INTERFACE I_NodeExecuteBeginEvent EXTENDS I_Event

PROPERTY PUBLIC TargetNode : I_Node
GET
END_GET
END_PROPERTY

END_INTERFACE

(* stored: Version 1.1.0.1, ProductVersion 3.1.4024.12
   Itf I_NodeExecuteBeginEvent: Id {aded8c3e-f1e0-0fb5-1926-ac2e0be4b934}
   Property TargetNode: Id {57165da3-ce42-039d-0de6-1c32b42a03db}
   Get Get: Id {6704add0-1f24-0633-09d9-7a070a45c4fe} *)
